// TIA Portal V16 export
// export: Created 2021-12-01T21:19:52.7260402Z, ExportSetting WithDefaults, DisplayName Totally Integrated Automation Portal, DisplayVersion V16 Update 4, DisplayName TIA Portal Version Control Interface, DisplayVersion V16 Update 2, DisplayName TIA Portal Openness, DisplayVersion V16 Update 4, DisplayName SINAMICS Startdrive Advanced, DisplayVersion V16 Update 5, DisplayName SINAMICS Startdrive G130, G150, S120, S150, SINAMICS MV, S210, DisplayVersion V16 Update 5, DisplayName SINAMICS Startdrive G110M, G120, G120C, G120D, G120P, G115D, DisplayVersion V16 Update 5, DisplayName STEP 7 Professional, DisplayVersion V16 Update 4, DisplayName STEP 7 Safety, DisplayVersion V16, DisplayName WinCC Advanced, DisplayVersion V16 Update 4
FUNCTION "ST00285_FC" : Void   // FC110, LAD
TITLE = ST00285
{ S7_Optimized_Access := 'TRUE' }
VERSION : 0.1
// stored: AutoNumber true, IsIECCheckEnabled false, SetENOAutomatically false, UDAEnableTagReadback false
   VAR_IN_OUT
      OPMODE : "OPMODE_OUT_UDT";
      HMI_EXTENSION : "HMI_EXTENSION_PANEL_UDT";
   END_VAR
   VAR_TEMP
      EmptyHS : "RT_HANDSHAKE_UDT";
   END_VAR
BEGIN

REGION Network 1: Alarm
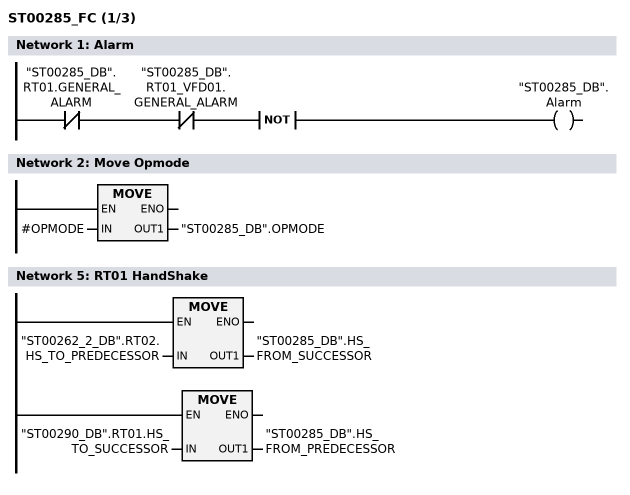
   RUNG wire#powerrail
      I_Contact( "ST00285_DB".RT01.GENERAL_ALARM )
      I_Contact( "ST00285_DB".RT01_VFD01.GENERAL_ALARM )
      Not()
      Coil( "ST00285_DB".Alarm )
   END_RUNG
   // the same network as SCL:
   "ST00285_DB".Alarm := NOT (NOT "ST00285_DB".RT01.GENERAL_ALARM AND NOT "ST00285_DB".RT01_VFD01.GENERAL_ALARM);
END_REGION

REGION Network 2: Move Opmode
   RUNG wire#powerrail
      Move(in := #OPMODE, out1 => "ST00285_DB".OPMODE)
   END_RUNG
   // the same network as SCL:
   "ST00285_DB".OPMODE := #OPMODE;
END_REGION

REGION Network 3: *******************RT01 Control*******************
END_REGION

REGION Network 4 (SCL): RT01 Parameters
   "ST00285_DB".RT01.PARA_SET.Para.PosEndForward1 := true;
   "ST00285_DB".RT01.PARA_SET.Para.PosEndReverse := true;
   "ST00285_DB".RT01.PARA_SET.Para.PosSlowForward := true;

   "ST00285_DB".RT01.PARA_SET.Set.RunTimeForward := 450;
   "ST00285_DB".RT01.PARA_SET.Set.RunTimeReverse := 450;
END_REGION

REGION Network 5: RT01 HandShake
   RUNG wire#powerrail
      Move(in := "ST00262_2_DB".RT02.HS_TO_PREDECESSOR, out1 => "ST00285_DB".HS_FROM_SUCCESSOR)
   END_RUNG
   RUNG wire#powerrail
      Move(in := "ST00290_DB".RT01.HS_TO_SUCCESSOR, out1 => "ST00285_DB".HS_FROM_PREDECESSOR)
   END_RUNG
   // the same network as SCL:
   "ST00285_DB".HS_FROM_SUCCESSOR := "ST00262_2_DB".RT02.HS_TO_PREDECESSOR;
   "ST00285_DB".HS_FROM_PREDECESSOR := "ST00290_DB".RT01.HS_TO_SUCCESSOR;
END_REGION

REGION Network 6: RT01 FB Control
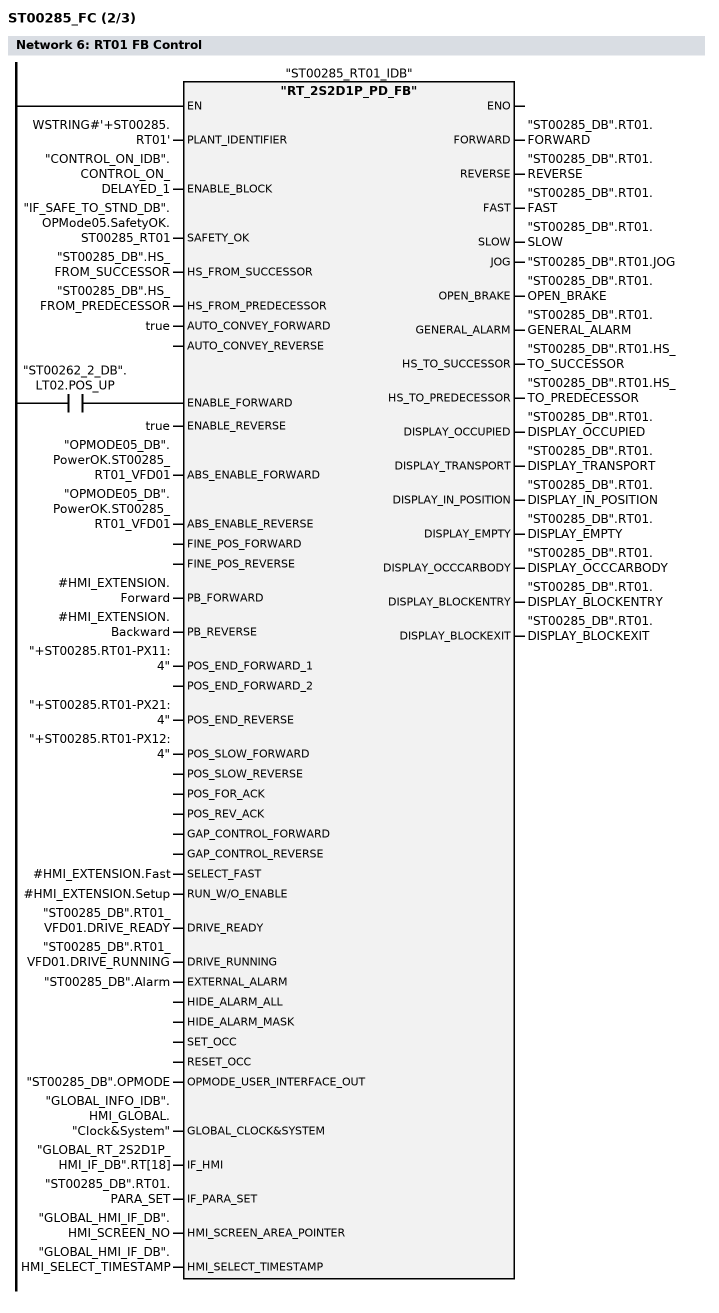
   RUNG wire#powerrail
      "ST00285_RT01_IDB"(ENABLE_FORWARD := wire#w1, PLANT_IDENTIFIER := WSTRING#'+ST00285.RT01', ENABLE_BLOCK := "CONTROL_ON_IDB".CONTROL_ON_DELAYED_1, SAFETY_OK := "IF_SAFE_TO_STND_DB".OPMode05.SafetyOK.ST00285_RT01, HS_FROM_SUCCESSOR := "ST00285_DB".HS_FROM_SUCCESSOR, HS_FROM_PREDECESSOR := "ST00285_DB".HS_FROM_PREDECESSOR, AUTO_CONVEY_FORWARD := true, AUTO_CONVEY_REVERSE :=, ENABLE_REVERSE := true, ABS_ENABLE_FORWARD := "OPMODE05_DB".PowerOK.ST00285_RT01_VFD01, ABS_ENABLE_REVERSE := "OPMODE05_DB".PowerOK.ST00285_RT01_VFD01, FINE_POS_FORWARD :=, FINE_POS_REVERSE :=, PB_FORWARD := #HMI_EXTENSION.Forward, PB_REVERSE := #HMI_EXTENSION.Backward, POS_END_FORWARD_1 := "+ST00285.RT01-PX11:4", POS_END_FORWARD_2 :=, POS_END_REVERSE := "+ST00285.RT01-PX21:4", POS_SLOW_FORWARD := "+ST00285.RT01-PX12:4", POS_SLOW_REVERSE :=, POS_FOR_ACK :=, POS_REV_ACK :=, GAP_CONTROL_FORWARD :=, GAP_CONTROL_REVERSE :=, SELECT_FAST := #HMI_EXTENSION.Fast, "RUN_W/O_ENABLE" := #HMI_EXTENSION.Setup, DRIVE_READY := "ST00285_DB".RT01_VFD01.DRIVE_READY, DRIVE_RUNNING := "ST00285_DB".RT01_VFD01.DRIVE_RUNNING, EXTERNAL_ALARM := "ST00285_DB".Alarm, HIDE_ALARM_ALL :=, HIDE_ALARM_MASK :=, SET_OCC :=, RESET_OCC :=, OPMODE_USER_INTERFACE_OUT := "ST00285_DB".OPMODE, "GLOBAL_CLOCK&SYSTEM" := "GLOBAL_INFO_IDB".HMI_GLOBAL."Clock&System", IF_HMI := "GLOBAL_RT_2S2D1P_HMI_IF_DB".RT[18], IF_PARA_SET := "ST00285_DB".RT01.PARA_SET, HMI_SCREEN_AREA_POINTER := "GLOBAL_HMI_IF_DB".HMI_SCREEN_NO, HMI_SELECT_TIMESTAMP := "GLOBAL_HMI_IF_DB".HMI_SELECT_TIMESTAMP, FORWARD => "ST00285_DB".RT01.FORWARD, REVERSE => "ST00285_DB".RT01.REVERSE, FAST => "ST00285_DB".RT01.FAST, SLOW => "ST00285_DB".RT01.SLOW, JOG => "ST00285_DB".RT01.JOG, OPEN_BRAKE => "ST00285_DB".RT01.OPEN_BRAKE, GENERAL_ALARM => "ST00285_DB".RT01.GENERAL_ALARM, HS_TO_SUCCESSOR => "ST00285_DB".RT01.HS_TO_SUCCESSOR, HS_TO_PREDECESSOR => "ST00285_DB".RT01.HS_TO_PREDECESSOR, DISPLAY_OCCUPIED => "ST00285_DB".RT01.DISPLAY_OCCUPIED, DISPLAY_TRANSPORT => "ST00285_DB".RT01.DISPLAY_TRANSPORT, DISPLAY_IN_POSITION => "ST00285_DB".RT01.DISPLAY_IN_POSITION, DISPLAY_EMPTY => "ST00285_DB".RT01.DISPLAY_EMPTY, DISPLAY_OCCCARBODY => "ST00285_DB".RT01.DISPLAY_OCCCARBODY, DISPLAY_BLOCKENTRY => "ST00285_DB".RT01.DISPLAY_BLOCKENTRY, DISPLAY_BLOCKEXIT => "ST00285_DB".RT01.DISPLAY_BLOCKEXIT)
   END_RUNG
   RUNG wire#powerrail
      Contact( "ST00262_2_DB".LT02.POS_UP )
   END_RUNG wire#w1
   // the same network as SCL:
   "ST00285_RT01_IDB"(PLANT_IDENTIFIER := WSTRING#'+ST00285.RT01',   // "RT_2S2D1P_PD_FB"
                      ENABLE_BLOCK := "CONTROL_ON_IDB".CONTROL_ON_DELAYED_1,
                      SAFETY_OK := "IF_SAFE_TO_STND_DB".OPMode05.SafetyOK.ST00285_RT01,
                      HS_FROM_SUCCESSOR := "ST00285_DB".HS_FROM_SUCCESSOR,
                      HS_FROM_PREDECESSOR := "ST00285_DB".HS_FROM_PREDECESSOR,
                      AUTO_CONVEY_FORWARD := true,
                      ENABLE_FORWARD := "ST00262_2_DB".LT02.POS_UP,
                      ENABLE_REVERSE := true,
                      ABS_ENABLE_FORWARD := "OPMODE05_DB".PowerOK.ST00285_RT01_VFD01,
                      ABS_ENABLE_REVERSE := "OPMODE05_DB".PowerOK.ST00285_RT01_VFD01,
                      PB_FORWARD := #HMI_EXTENSION.Forward,
                      PB_REVERSE := #HMI_EXTENSION.Backward,
                      POS_END_FORWARD_1 := "+ST00285.RT01-PX11:4",
                      POS_END_REVERSE := "+ST00285.RT01-PX21:4",
                      POS_SLOW_FORWARD := "+ST00285.RT01-PX12:4",
                      SELECT_FAST := #HMI_EXTENSION.Fast,
                      "RUN_W/O_ENABLE" := #HMI_EXTENSION.Setup,
                      DRIVE_READY := "ST00285_DB".RT01_VFD01.DRIVE_READY,
                      DRIVE_RUNNING := "ST00285_DB".RT01_VFD01.DRIVE_RUNNING,
                      EXTERNAL_ALARM := "ST00285_DB".Alarm,
                      OPMODE_USER_INTERFACE_OUT := "ST00285_DB".OPMODE,
                      "GLOBAL_CLOCK&SYSTEM" := "GLOBAL_INFO_IDB".HMI_GLOBAL."Clock&System",
                      IF_HMI := "GLOBAL_RT_2S2D1P_HMI_IF_DB".RT[18],
                      IF_PARA_SET := "ST00285_DB".RT01.PARA_SET,
                      HMI_SCREEN_AREA_POINTER := "GLOBAL_HMI_IF_DB".HMI_SCREEN_NO,
                      HMI_SELECT_TIMESTAMP := "GLOBAL_HMI_IF_DB".HMI_SELECT_TIMESTAMP,
                      FORWARD => "ST00285_DB".RT01.FORWARD,
                      REVERSE => "ST00285_DB".RT01.REVERSE,
                      FAST => "ST00285_DB".RT01.FAST,
                      SLOW => "ST00285_DB".RT01.SLOW,
                      JOG => "ST00285_DB".RT01.JOG,
                      OPEN_BRAKE => "ST00285_DB".RT01.OPEN_BRAKE,
                      GENERAL_ALARM => "ST00285_DB".RT01.GENERAL_ALARM,
                      HS_TO_SUCCESSOR => "ST00285_DB".RT01.HS_TO_SUCCESSOR,
                      HS_TO_PREDECESSOR => "ST00285_DB".RT01.HS_TO_PREDECESSOR,
                      DISPLAY_OCCUPIED => "ST00285_DB".RT01.DISPLAY_OCCUPIED,
                      DISPLAY_TRANSPORT => "ST00285_DB".RT01.DISPLAY_TRANSPORT,
                      DISPLAY_IN_POSITION => "ST00285_DB".RT01.DISPLAY_IN_POSITION,
                      DISPLAY_EMPTY => "ST00285_DB".RT01.DISPLAY_EMPTY,
                      DISPLAY_OCCCARBODY => "ST00285_DB".RT01.DISPLAY_OCCCARBODY,
                      DISPLAY_BLOCKENTRY => "ST00285_DB".RT01.DISPLAY_BLOCKENTRY,
                      DISPLAY_BLOCKEXIT => "ST00285_DB".RT01.DISPLAY_BLOCKEXIT);
END_REGION

REGION Network 7: RT01 Speed
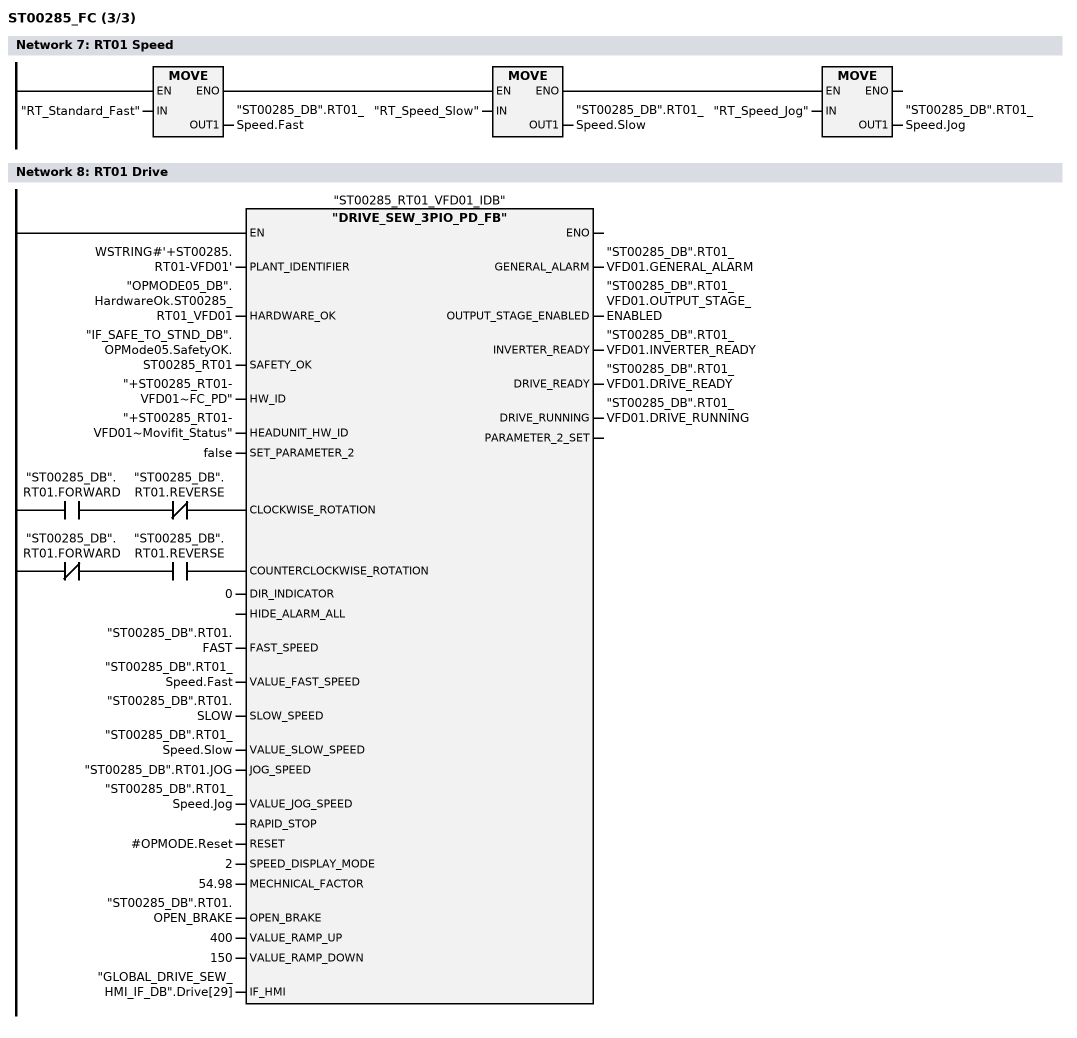
   RUNG wire#powerrail
      Move(in := "RT_Standard_Fast", out1 => "ST00285_DB".RT01_Speed.Fast)
      Move(in := "RT_Speed_Slow", out1 => "ST00285_DB".RT01_Speed.Slow)
      Move(in := "RT_Speed_Jog", out1 => "ST00285_DB".RT01_Speed.Jog)
   END_RUNG
   // the same network as SCL:
   "ST00285_DB".RT01_Speed.Fast := "RT_Standard_Fast";
   "ST00285_DB".RT01_Speed.Slow := "RT_Speed_Slow";
   "ST00285_DB".RT01_Speed.Jog := "RT_Speed_Jog";
END_REGION

REGION Network 8: RT01 Drive
   RUNG wire#powerrail
      "ST00285_RT01_VFD01_IDB"(CLOCKWISE_ROTATION := wire#w1, COUNTERCLOCKWISE_ROTATION := wire#w2, PLANT_IDENTIFIER := WSTRING#'+ST00285.RT01-VFD01', HARDWARE_OK := "OPMODE05_DB".HardwareOk.ST00285_RT01_VFD01, SAFETY_OK := "IF_SAFE_TO_STND_DB".OPMode05.SafetyOK.ST00285_RT01, HW_ID := "+ST00285_RT01-VFD01~FC_PD", HEADUNIT_HW_ID := "+ST00285_RT01-VFD01~Movifit_Status", SET_PARAMETER_2 := false, DIR_INDICATOR := 0, HIDE_ALARM_ALL :=, FAST_SPEED := "ST00285_DB".RT01.FAST, VALUE_FAST_SPEED := "ST00285_DB".RT01_Speed.Fast, SLOW_SPEED := "ST00285_DB".RT01.SLOW, VALUE_SLOW_SPEED := "ST00285_DB".RT01_Speed.Slow, JOG_SPEED := "ST00285_DB".RT01.JOG, VALUE_JOG_SPEED := "ST00285_DB".RT01_Speed.Jog, RAPID_STOP :=, RESET := #OPMODE.Reset, SPEED_DISPLAY_MODE := 2, MECHNICAL_FACTOR := 54.98, OPEN_BRAKE := "ST00285_DB".RT01.OPEN_BRAKE, VALUE_RAMP_UP := 400, VALUE_RAMP_DOWN := 150, IF_HMI := "GLOBAL_DRIVE_SEW_HMI_IF_DB".Drive[29], GENERAL_ALARM => "ST00285_DB".RT01_VFD01.GENERAL_ALARM, OUTPUT_STAGE_ENABLED => "ST00285_DB".RT01_VFD01.OUTPUT_STAGE_ENABLED, INVERTER_READY => "ST00285_DB".RT01_VFD01.INVERTER_READY, DRIVE_READY => "ST00285_DB".RT01_VFD01.DRIVE_READY, DRIVE_RUNNING => "ST00285_DB".RT01_VFD01.DRIVE_RUNNING, PARAMETER_2_SET =>)
   END_RUNG
   RUNG wire#powerrail
      Contact( "ST00285_DB".RT01.FORWARD )
      I_Contact( "ST00285_DB".RT01.REVERSE )
   END_RUNG wire#w1
   RUNG wire#powerrail
      I_Contact( "ST00285_DB".RT01.FORWARD )
      Contact( "ST00285_DB".RT01.REVERSE )
   END_RUNG wire#w2
   // the same network as SCL:
   "ST00285_RT01_VFD01_IDB"(PLANT_IDENTIFIER := WSTRING#'+ST00285.RT01-VFD01',   // "DRIVE_SEW_3PIO_PD_FB"
                           HARDWARE_OK := "OPMODE05_DB".HardwareOk.ST00285_RT01_VFD01,
                           SAFETY_OK := "IF_SAFE_TO_STND_DB".OPMode05.SafetyOK.ST00285_RT01,
                           HW_ID := "+ST00285_RT01-VFD01~FC_PD",
                           HEADUNIT_HW_ID := "+ST00285_RT01-VFD01~Movifit_Status",
                           SET_PARAMETER_2 := false,
                           CLOCKWISE_ROTATION := "ST00285_DB".RT01.FORWARD AND NOT "ST00285_DB".RT01.REVERSE,
                           COUNTERCLOCKWISE_ROTATION := NOT "ST00285_DB".RT01.FORWARD AND "ST00285_DB".RT01.REVERSE,
                           DIR_INDICATOR := 0,
                           FAST_SPEED := "ST00285_DB".RT01.FAST,
                           VALUE_FAST_SPEED := "ST00285_DB".RT01_Speed.Fast,
                           SLOW_SPEED := "ST00285_DB".RT01.SLOW,
                           VALUE_SLOW_SPEED := "ST00285_DB".RT01_Speed.Slow,
                           JOG_SPEED := "ST00285_DB".RT01.JOG,
                           VALUE_JOG_SPEED := "ST00285_DB".RT01_Speed.Jog,
                           RESET := #OPMODE.Reset,
                           SPEED_DISPLAY_MODE := 2,
                           MECHNICAL_FACTOR := 54.98,
                           OPEN_BRAKE := "ST00285_DB".RT01.OPEN_BRAKE,
                           VALUE_RAMP_UP := 400,
                           VALUE_RAMP_DOWN := 150,
                           IF_HMI := "GLOBAL_DRIVE_SEW_HMI_IF_DB".Drive[29],
                           GENERAL_ALARM => "ST00285_DB".RT01_VFD01.GENERAL_ALARM,
                           OUTPUT_STAGE_ENABLED => "ST00285_DB".RT01_VFD01.OUTPUT_STAGE_ENABLED,
                           INVERTER_READY => "ST00285_DB".RT01_VFD01.INVERTER_READY,
                           DRIVE_READY => "ST00285_DB".RT01_VFD01.DRIVE_READY,
                           DRIVE_RUNNING => "ST00285_DB".RT01_VFD01.DRIVE_RUNNING);
END_REGION
END_FUNCTION
